// Mitsubishi GX Works2 project: replay1   PLC: Q03UDV

PROGRAM MAIN
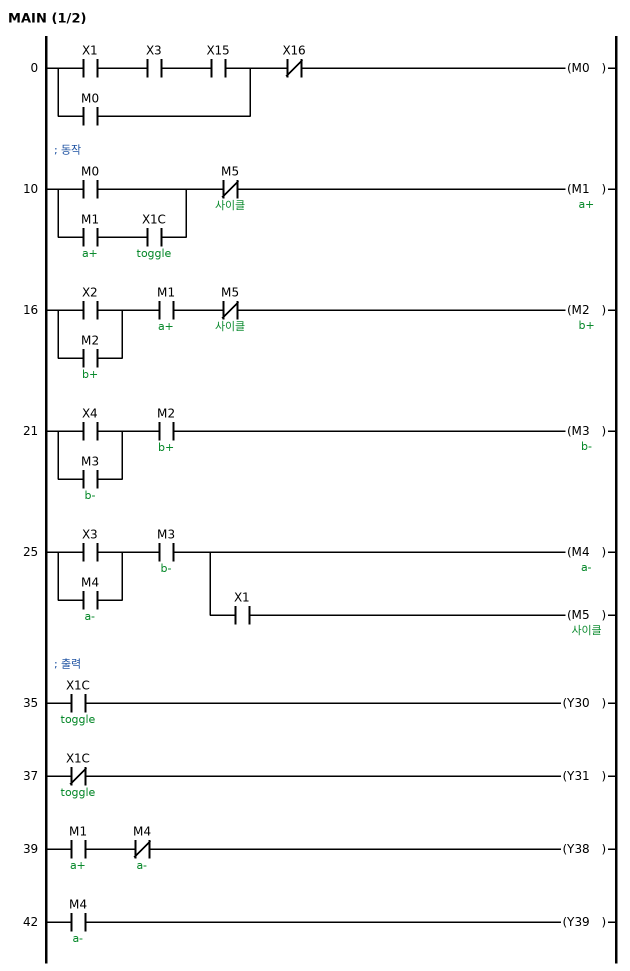
0     LD      X1
      AND     X3
      AND     X15
      OR      M0
      ANI     X16
      OUT     M0
; 동작
10    LD      M0
      LD      M1  ; a+
      AND     X1C  ; toggle
      ORB
      ANI     M5  ; 사이클
      OUT     M1  ; a+
16    LD      X2
      OR      M2  ; b+
      AND     M1  ; a+
      ANI     M5  ; 사이클
      OUT     M2  ; b+
21    LD      X4
      OR      M3  ; b-
      AND     M2  ; b+
      OUT     M3  ; b-
25    LD      X3
      OR      M4  ; a-
      AND     M3  ; b-
      OUT     M4  ; a-
      AND     X1
      OUT     M5  ; 사이클
; 출력
35    LD      X1C  ; toggle
      OUT     Y30
37    LDI     X1C  ; toggle
      OUT     Y31
39    LD      M1  ; a+
      ANI     M4  ; a-
      OUT     Y38
42    LD      M4  ; a-
      OUT     Y39
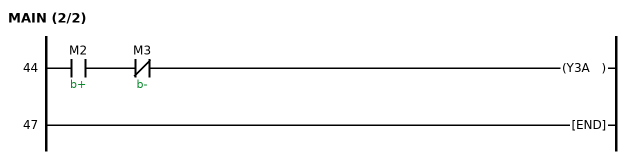
44    LD      M2  ; b+
      ANI     M3  ; b-
      OUT     Y3A
47    END
END_PROGRAM
